(* CODESYS project SingleElevator.project

Project tree, tasks and I/O mapping:
  Device : CODESYS Control Win V3, 3S - Smart Software Solutions GmbH, version 3.5.16.20
    application Application
      libraries: Standard, * (System)
      task MainTask (cyclic, interval t#20ms, priority 1) calls Simulation, GAinstances, PLC_PRG
      task VISU_TASK (cyclic, interval 100 ms, priority 31) calls VisuElems.Visu_Prg
      global variables GVL
      visualisation Visualization
      program Simulation [ST]
      program GAinstances [FBD]
      program PLC_PRG [SFC]: Closing_active, Closing_exit, CloseDoors2_exit, CloseDoors_active, CloseDoors_exit, FirstFloor_active, FirstFloor_exit, OpenDoors_active, OpenDoors_exit, CloseDoors2_active, Destination_active, Destination_exit, OpenDoors2_active, OpenDoors2_exit, WaitForCalls_active, PreCalls_active, MidCalls_active, MidCalls_entry, WaitForCalls_exit, PreCalls_entry, Dummy4_exit, LEDActive_active, LEDnotActive_active, GetCalls_active, FirstFloor_entry, Destination_entry
      GA/
        function block Doors_GA [SFC]: Init_active, Ready_active, Busy_active
        function block Motoring_GA [SFC]: Init_active, Ready_active, Busy_active, StartMotor_active, HighSpeed_active, StartGoDown_active, StartGoDown_exit, GroundFloor_active, GroundFloor_exit, LowSpeed_active, LowSpeed_exit, CountingDecks_active, Working_active, Extremes_active, Extremes_exit, Extremes_entry, StartMotor_exit
  text list GlobalTextList
*)

// Device/Application/GVL
{attribute 'qualified_only'}
VAR_GLOBAL
	ManageDoors: Doors_GA;
	Motoring : Motoring_GA;
	
(* Elevator managing variables*)
	Open: BOOL;				(* Sensor: the door is fully open*)
	Closed: BOOL;			(* Sensor: the door is fully closed*)
	LimitDown: BOOL;		(* Sensor: lower limit sensor, if TRUE the lift has reached the lower limit*)
	LimitUp: BOOL;			(* Sensor: upper limit sensor, if TRUE the lift has reached the upper limit*)
	DeckSensor: BOOL;		(* Sensor: if TRUE the cab is in proximity of a deck*)
	RampSensor: BOOL;		(* Sensor: if TRUE the cab is in proximity of a ramp*)
	Presence :BOOL; 		(* Sensor: if TRUE something blocks the door photocell*)
	Emergency: BOOL;		(* Input: if TRUE the emergency button has been pressed*)

	Closing: BOOL;			(* Actuator: if TRUE the door starts closing*)
	Opening: BOOL;			(* Actuator: the door starts opening*)
	Motor_on: BOOL;			(* Actuator: if TRUE the lift pulley motor start moving*)
	Up: BOOL;				(* Actuator parameter: if TRUE the lift moves upward, downward otherwise*)
	Vel: BOOL;				(* Actuator parameter: motor speed, if TRUE high speed, low speed otherwise*)


	Current: INT;  			(* Visualization: variable used to storage the current deck*)
    Destination: INT;		(* Visualization: variable used to storage the the destination deck*)
	EmergencyVis: BOOL; 	(* Visualization: if TRUE the emergency light is turned on*)

	InitialDeck: INT := 1;	(* Only for simulation: variable used to define the initial deck*)
	InitCycle: BOOL := FALSE;(* Only for simulation: used to execute the instruction at the first cycle*)
	Height: INT;			(* Only for simulation: elevator height*)
	DeckRest: INT;        	(* Only for simulation: division rest for generating deck sensor*)
	Memory: INT;
	RampRest: INT;			(* Only for simulation: division rest for generating the ramp position*)
	MemoryR: INT;
	Door: INT;				(* Only for simulation: to visualize the closing of the door*)
	Displacement: INT;		(* Only for simulation: lift displacement, dependent on the motor speed*)

 (*Inputs: internal panel variables*)
	PG: BOOL;
	P1: BOOL;
	P2: BOOL;
	P3: BOOL;
	P4: BOOL;
	P5: BOOL;
	P6: BOOL;
	P7: BOOL;

(*Visualization: internal panel variables used to turn on the LED*)
	PGVis: BOOL;
	P1Vis: BOOL;
	P2Vis: BOOL;
	P3Vis: BOOL;
	P4Vis: BOOL;
	P5Vis: BOOL;
	P6Vis: BOOL;
	P7Vis: BOOL;

(*Inputs: external panel variables*)
	UpDeckG: BOOL;
	UpDeck1: BOOL;
	UpDeck2: BOOL;
	UpDeck3: BOOL;
	UpDeck4: BOOL;
	UpDeck5: BOOL;
	UpDeck6: BOOL;
	DownDeck7: BOOL;
	DownDeck6: BOOL;
	DownDeck5: BOOL;
	DownDeck4: BOOL;
	DownDeck3: BOOL;
	DownDeck2: BOOL;
	DownDeck1: BOOL;

(*Visualization: external panel variables used to turn on the LED*)
	UpDeckGVis: BOOL;
	UpDeck1Vis: BOOL;
	UpDeck2Vis: BOOL;
	UpDeck3Vis: BOOL;
	UpDeck4Vis: BOOL;
	UpDeck5Vis: BOOL;
	UpDeck6Vis: BOOL;
	DownDeck7Vis: BOOL;
	DownDeck6Vis: BOOL;
	DownDeck5Vis: BOOL;
	DownDeck4Vis: BOOL;
	DownDeck3Vis: BOOL;
	DownDeck2Vis: BOOL;
	DownDeck1Vis: BOOL;

(*Only for simulation: variables used to simulate the fault on deck sensor*)
	SensorG: BOOL;				(* if TRUE the magnetic information for deck G is lost and the deck sensor cannot become TRUE*)
	Sensor1: BOOL;				(* if TRUE the magnetic information for deck 1 is lost and the deck sensor cannot become TRUE*)
	Sensor2: BOOL;
	Sensor3: BOOL;
	Sensor4: BOOL;
	Sensor5: BOOL;
	Sensor6: BOOL;
	Sensor7: BOOL;
	FaultSensorAlarm: BOOL; 	(* Visulaization: if TRUE alerts the user of a deck sensor fault*)

(*Only for simulation: variables used to simulate the fault on ramp sensor*)
	RampGUp: BOOL;
	Ramp1Down: BOOL;
	Ramp1Up:BOOL;
	Ramp2Down: BOOL;
	Ramp2Up:BOOL;
	Ramp3Down: BOOL;
	Ramp3Up:BOOL;
	Ramp4Down: BOOL;
	Ramp4Up:BOOL;
	Ramp5Down: BOOL;
	Ramp5Up:BOOL;
	Ramp6Down: BOOL;
	Ramp6Up:BOOL;
	Ramp7Down: BOOL;
	FaultRampAlarm: BOOL; 		(* Visulaization: if TRUE alerts the user of a ramp sensor fault*)
	SensorGOK: BOOL;
	Sensor1OK: BOOL;
	Sensor2OK: BOOL;
	Sensor6OK: BOOL;
	Sensor3OK: BOOL;
	Sensor4OK: BOOL;
	Sensor5OK: BOOL;
	Sensor7OK: BOOL;
	RampGUpOK: BOOL;
	Ramp1DownOK: BOOL;
	Ramp1UpOK: BOOL;
	Ramp2DownOK: BOOL;
	Ramp2UpOK: BOOL;
	Ramp3DownOK: BOOL;
	Ramp3UpOK: BOOL;
	Ramp4DownOK: BOOL;
	Ramp4UpOK: BOOL;
	Ramp5DownOK: BOOL;
	Ramp5UpOK: BOOL;
	Ramp6DownOK: BOOL;
	Ramp6UpOK: BOOL;
	Ramp7DownOK: BOOL;
	Ramp7UpOK: BOOL;
END_VAR

// Device/Application/Simulation
PROGRAM Simulation
VAR
END_VAR

(* Initial position of the cab inside the hoistway. It is executed only at the first cycle.  *)
IF NOT GVL.InitCycle THEN
			GVL.InitCycle := TRUE ;
			GVL.Height := 20 * GVL.InitialDeck;
		    GVL.Door := 0;
			GVL.Current := GVL.Height / 20;
END_IF;

(* Elevator management, these instructions are executed each cycle time*)

(* Elevator door control. *)
IF GVL.Closing THEN
	GVL.Door := GVL.Door + 1;		(*Closing door management*)
	GVL.Open := FALSE;
END_IF

IF GVL.Door >= 60 THEN						(* Closed door limit*)
	GVL.Closed := TRUE;
END_IF

IF GVL.Opening THEN
	GVL.Door := GVL.Door - 1; 	(* Opening door management*)
	GVL.Closed := FALSE;
END_IF

IF GVL.Door <= 0 THEN							(* Open door limit*)
	GVL.Open := TRUE;
END_IF


(* Maximum and minimum management in the door simulation*)
IF GVL.Door < 0 THEN
	 GVL.Door := 0;
END_IF

IF GVL.Door > 60 THEN
	GVL.Door := 60;
END_IF


(* Control of the cab position inside the hostway. *)
(* Displacement definition for graphic visualization*)
IF GVL.Vel THEN 
	GVL.Displacement := 2;
ELSE 
	GVL.Displacement := 1;
END_IF


(* Height modification relying on direction and speed*)
IF GVL.Motor_on AND GVL.Up THEN
	GVL.Height := GVL.Height + GVL.Displacement;
	GVL.LimitDown := FALSE;
END_IF

IF GVL.Motor_on AND NOT GVL.Up THEN
	GVL.Height := GVL.Height - GVL.Displacement;
	GVL.LimitUp := FALSE;
END_IF


(* Limits for visualization*)
IF GVL.Height < -20 THEN
	GVL.Height := -20;
END_IF

IF GVL.Height > 160 THEN
	GVL.Height := 160;
END_IF

(* Limit sensors management*)
IF GVL.Height <= -10 THEN
	GVL.LimitDown := TRUE;
END_IF

IF GVL.Height >= 150 THEN
	 GVL.LimitUp := TRUE;
END_IF


(*-------------------------------------------------------------------*)
(*  Fault Management (Deck and Ramp Sensors)   *)
(*-------------------------------------------------------------------*)
(* Deck Sensor*)
(* Range of value where the deck sensor is active*)
IF ((GVL.Height >= -1) AND (GVL.Height <= 1)) THEN
	GVL.SensorGOK := TRUE;
ELSE  
	GVL.SensorGOK := FALSE;
END_IF

IF ((GVL.Height >= 20-1) AND (GVL.Height <= 20+1)) THEN
	GVL.Sensor1OK := TRUE;
ELSE  
	GVL.Sensor1OK := FALSE;
END_IF

IF ((GVL.Height >= 40-1) AND (GVL.Height <= 40+1)) THEN
	GVL.Sensor2OK := TRUE;
ELSE  
	GVL.Sensor2OK := FALSE;
END_IF

IF ((GVL.Height >= 60-1) AND (GVL.Height <= 60+1)) THEN
	GVL.Sensor3OK := TRUE;
ELSE  
	GVL.Sensor3OK := FALSE;
END_IF

IF ((GVL.Height >= 80-1) AND (GVL.Height <= 80+1)) THEN
	GVL.Sensor4OK := TRUE;
ELSE  
	GVL.Sensor4OK := FALSE;
END_IF

IF ((GVL.Height >= 100-1) AND (GVL.Height <= 100+1)) THEN
	GVL.Sensor5OK := TRUE;
ELSE   
	GVL.Sensor5OK := FALSE;
END_IF

IF ((GVL.Height >= 120-1) AND (GVL.Height <= 120+1)) THEN
	GVL.Sensor6OK := TRUE;
ELSE  
	GVL.Sensor6OK := FALSE;
END_IF

IF ((GVL.Height >= 140-1) AND (GVL.Height <= 140+1)) THEN
	GVL.Sensor7OK := TRUE;
ELSE  
	GVL.Sensor7OK := FALSE;
END_IF

GVL.DeckSensor := (GVL.SensorGOK AND NOT GVL.SensorG) OR
				    (GVL.Sensor1OK AND NOT GVL.Sensor1) OR
				    (GVL.Sensor2OK AND NOT GVL.Sensor2) OR
				    (GVL.Sensor3OK AND NOT GVL.Sensor3) OR
				    (GVL.Sensor4OK AND NOT GVL.Sensor4) OR
				    (GVL.Sensor5OK AND NOT GVL.Sensor5) OR
				    (GVL.Sensor6OK AND NOT GVL.Sensor6) OR
				    (GVL.Sensor7OK AND NOT GVL.Sensor7);

(* Ramp Sensor*)
(* Range of value where the ramp sensor is active*)
IF ((GVL.Height >= 5-1) AND (GVL.Height <= 5+1)) THEN
	GVL.RampGUpOK := TRUE;
ELSE 
	GVL.RampGUpOK := FALSE;
END_IF

(* Ramp close to deck 1*)
IF ((GVL.Height >= 15-1) AND (GVL.Height <= 15+1)) THEN
	GVL.Ramp1DownOK := TRUE;
ELSE 
	GVL.Ramp1DownOK := FALSE;
END_IF

IF ((GVL.Height >= 25-1) AND (GVL.Height <= 25+1)) THEN
	GVL.Ramp1UpOK := TRUE;
ELSE 
	GVL.Ramp1UpOK := FALSE;
END_IF

(* Ramp close to deck 2*)
IF ((GVL.Height >= 35-1) AND (GVL.Height <= 35+1)) THEN
	GVL.Ramp2DownOK := TRUE;
ELSE 
	GVL.Ramp2DownOK := FALSE;
END_IF

IF ((GVL.Height >= 45-1) AND (GVL.Height <= 45+1)) THEN
	GVL.Ramp2UpOK := TRUE;
ELSE 
	GVL.Ramp2UpOK := FALSE;
END_IF

(*Ramp close to deck  3*)
IF ((GVL.Height >= 55-1) AND (GVL.Height <= 55+1)) THEN
	GVL.Ramp3DownOK := TRUE;
ELSE 
	GVL.Ramp3DownOK := FALSE;
END_IF

IF ((GVL.Height >= 65-1) AND (GVL.Height <= 65+1)) THEN
	GVL.Ramp3UpOK := TRUE;
ELSE 
	GVL.Ramp3UpOK := FALSE;
END_IF

(* Ramp close to deck  4*)
IF ((GVL.Height >= 75-1) AND (GVL.Height <= 75+1)) THEN
	GVL.Ramp4DownOK := TRUE;
ELSE 
	GVL.Ramp4DownOK := FALSE;
END_IF

IF ((GVL.Height >= 85-1) AND (GVL.Height <= 85+1)) THEN
	GVL.Ramp4UpOK := TRUE;
ELSE 
	GVL.Ramp4UpOK:=FALSE;
END_IF

(* Ramp close to deck  5*)
IF ((GVL.Height >= 95-1) AND (GVL.Height <= 95+1)) THEN
	GVL.Ramp5DownOK := TRUE;
ELSE 
	GVL.Ramp5DownOK := FALSE;
END_IF

IF ((GVL.Height >= 105-1) AND (GVL.Height <= 105+1)) THEN
	GVL.Ramp5UpOK := TRUE;
ELSE
	GVL.Ramp5UpOK := FALSE;
END_IF

(* Ramp close to deck  6*)
IF ((GVL.Height >= 115-1) AND (GVL.Height <= 115+1)) THEN
	GVL.Ramp6DownOK := TRUE;
ELSE 
	GVL.Ramp6DownOK := FALSE;
END_IF

IF ((GVL.Height >= 125-1) AND (GVL.Height <= 125+1)) THEN
	GVL.Ramp6UpOK := TRUE;
ELSE 
	GVL.Ramp6UpOK := FALSE;
END_IF

(* Ramp close to deck  7*)
IF ((GVL.Height >= 135-1) AND (GVL.Height <= 135+1)) THEN
	GVL.Ramp7DownOK := TRUE;
ELSE 
	GVL.Ramp7DownOK := FALSE;
END_IF

GVL.RampSensor:=(GVL.RampGUpOK AND NOT GVL.RampGUp) OR 
								(GVL.Ramp1DownOK AND NOT GVL.Ramp1Down ) OR 
								(GVL.Ramp1UpOK AND NOT GVL.Ramp1Up ) OR
								(GVL.Ramp2DownOK AND NOT GVL.Ramp2Down ) OR 
								(GVL.Ramp2UpOK AND NOT GVL.Ramp2Up ) OR
								(GVL.Ramp3DownOK AND NOT GVL.Ramp3Down ) OR
 								(GVL.Ramp3UpOK AND NOT GVL.Ramp3Up ) OR
								(GVL.Ramp4DownOK AND NOT GVL.Ramp4Down ) OR
 								(GVL.Ramp4UpOK AND NOT GVL.Ramp4Up ) OR
								(GVL.Ramp5DownOK AND NOT GVL.Ramp5Down ) OR
 								(GVL.Ramp5UpOK AND NOT GVL.Ramp5Up ) OR
								(GVL.Ramp6DownOK AND NOT GVL.Ramp6Down ) OR
								(GVL.Ramp6UpOK AND NOT GVL.Ramp6Up ) OR
								(GVL.Ramp7DownOK AND NOT GVL.Ramp7Down );

END_PROGRAM

// Device/Application/GAinstances
PROGRAM GAinstances
VAR
END_VAR

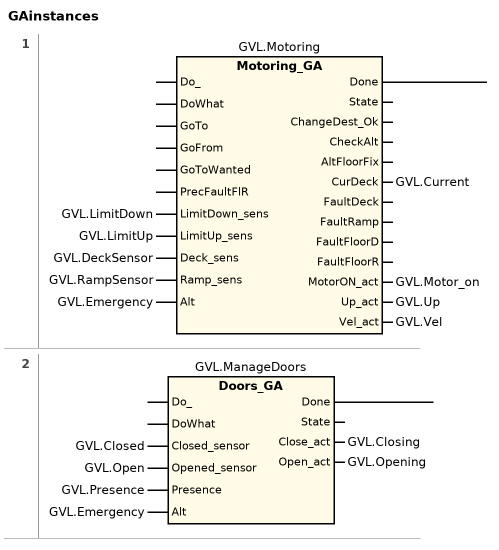
// NETWORK 1
GVL.Motoring(
    LimitDown_sens := GVL.LimitDown,
    LimitUp_sens := GVL.LimitUp,
    Deck_sens := GVL.DeckSensor,
    Ramp_sens := GVL.RampSensor,
    Alt := GVL.Emergency,
    CurDeck => GVL.Current,
    MotorON_act => GVL.Motor_on,
    Up_act => GVL.Up,
    Vel_act => GVL.Vel); // Motoring_GA

// NETWORK 2
GVL.ManageDoors(
    Closed_sensor := GVL.Closed,
    Opened_sensor := GVL.Open,
    Presence := GVL.Presence,
    Alt := GVL.Emergency,
    Close_act => GVL.Closing,
    Open_act => GVL.Opening); // Doors_GA

END_PROGRAM

// Device/Application/GA/Motoring_GA
FUNCTION_BLOCK Motoring_GA
VAR_INPUT
	Do_: BOOL;
	DoWhat: STRING;
	GoTo: INT;
	GoFrom: INT;
	GoToWanted: INT;
	PrecFaultFlR: ARRAY[0..7] OF INT;
	
	//SENSORS
	LimitDown_sens: BOOL;
	LimitUp_sens: BOOL;
	Deck_sens: BOOL;
	Ramp_sens: BOOL;
	
	Alt: BOOL;
END_VAR

VAR_OUTPUT
	Done: BOOL;
	State: STRING;
	ChangeDest_Ok: BOOL;
	CheckAlt: BOOL;
	AltFloorFix: INT;
	CurDeck: INT;
	
	//FAULTS
	FaultDeck: BOOL;
	FaultRamp: BOOL;
	FaultFloorD: ARRAY[0..7] OF INT;
	FaultFloorR: ARRAY[0..7] OF INT;
	
	//ACTUATORS
	MotorON_act: BOOL;
	Up_act: BOOL;
	Vel_act: BOOL;
END_VAR
VAR
	i: INT;
	Cont: INT;
	CheckRamps: BOOL;
	Initial: BOOL;
	
	AltFloor: INT;
	Fault: BOOL;
	Faults: ARRAY[0..21] OF BOOL;
	DeckPrec: INT;
	RampPrec: INT;
	FirstTime: BOOL;
	TrueFault: INT;
	NoProbFault: BOOL;
	FaultSameD: BOOL;
	SecondRamp: BOOL;
	Down_sens: BOOL;
	Up_sens: BOOL;
	CorrDone: BOOL;
	Sens: BOOL;
END_VAR

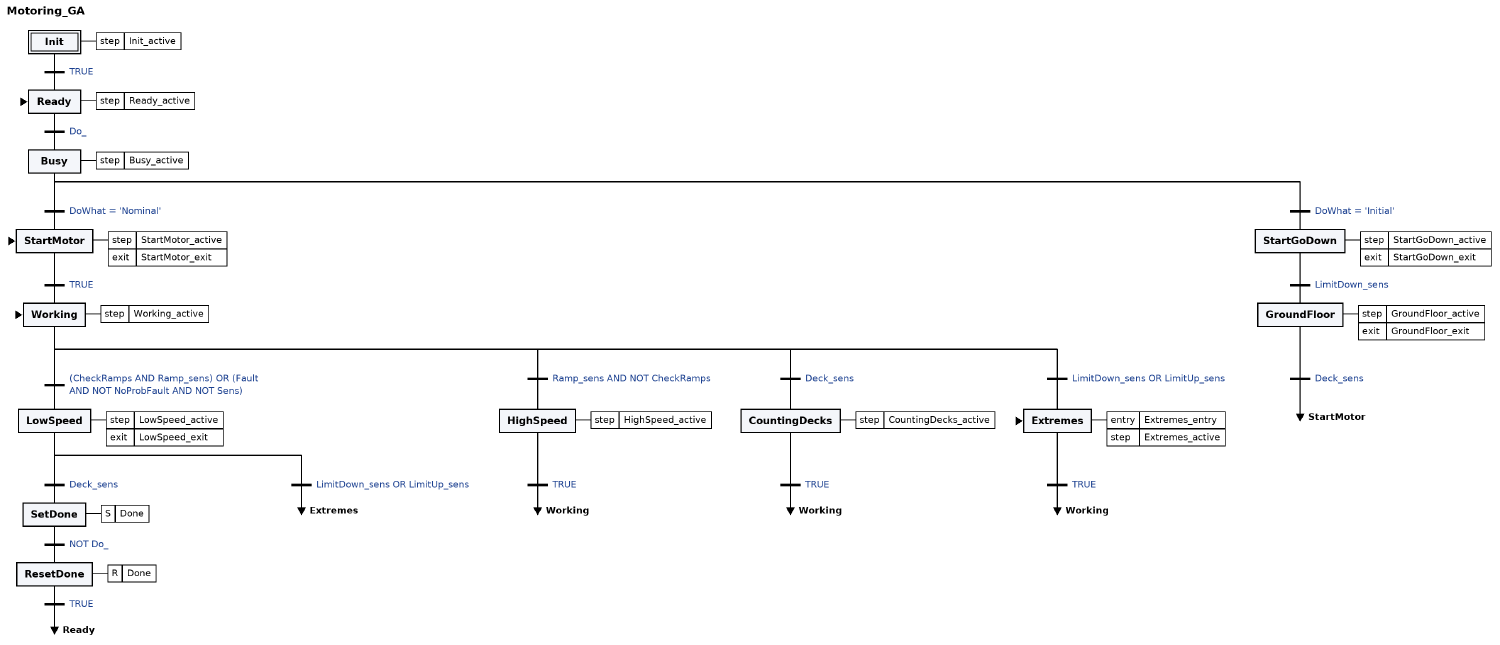
INITIAL_STEP Init:
    Init_active(N);  // step action
END_STEP
TRANSITION FROM Init TO Ready
    := TRUE;
END_TRANSITION
STEP Ready:
    Ready_active(N);  // step action
END_STEP
TRANSITION FROM Ready TO Busy
    := Do_;
END_TRANSITION
STEP Busy:
    Busy_active(N);  // step action
END_STEP
TRANSITION FROM Busy TO StartMotor
    := DoWhat = 'Nominal';
END_TRANSITION
STEP StartMotor:
    StartMotor_active(N);  // step action
    StartMotor_exit(P0);  // exit action
END_STEP
TRANSITION FROM StartMotor TO Working
    := TRUE;
END_TRANSITION
STEP Working:
    Working_active(N);  // step action
END_STEP
TRANSITION FROM Working TO LowSpeed
    := (CheckRamps AND Ramp_sens) OR (Fault AND NOT NoProbFault AND NOT Sens);
END_TRANSITION
STEP LowSpeed:
    LowSpeed_active(N);  // step action
    LowSpeed_exit(P0);  // exit action
END_STEP
TRANSITION FROM Working TO HighSpeed
    := Ramp_sens AND NOT CheckRamps;
END_TRANSITION
STEP HighSpeed:
    HighSpeed_active(N);  // step action
END_STEP
TRANSITION FROM HighSpeed TO Working
    := TRUE;
END_TRANSITION
TRANSITION FROM Working TO CountingDecks
    := Deck_sens;
END_TRANSITION
STEP CountingDecks:
    CountingDecks_active(N);  // step action
END_STEP
TRANSITION FROM CountingDecks TO Working
    := TRUE;
END_TRANSITION
TRANSITION FROM Working TO Extremes
    := LimitDown_sens OR LimitUp_sens;
END_TRANSITION
STEP Extremes:
    Extremes_entry(P1);  // entry action
    Extremes_active(N);  // step action
END_STEP
TRANSITION FROM Extremes TO Working
    := TRUE;
END_TRANSITION
TRANSITION FROM LowSpeed TO SetDone
    := Deck_sens;
END_TRANSITION
TRANSITION FROM LowSpeed TO Extremes
    := LimitDown_sens OR LimitUp_sens;
END_TRANSITION
TRANSITION FROM Busy TO StartGoDown
    := DoWhat = 'Initial';
END_TRANSITION
STEP StartGoDown:
    StartGoDown_active(N);  // step action
    StartGoDown_exit(P0);  // exit action
END_STEP
TRANSITION FROM StartGoDown TO GroundFloor
    := LimitDown_sens;
END_TRANSITION
STEP GroundFloor:
    GroundFloor_active(N);  // step action
    GroundFloor_exit(P0);  // exit action
END_STEP
TRANSITION FROM GroundFloor TO StartMotor
    := Deck_sens;
END_TRANSITION
STEP SetDone:
    Done(S);
END_STEP
TRANSITION FROM SetDone TO ResetDone
    := NOT Do_;
END_TRANSITION
STEP ResetDone:
    Done(R);
END_STEP
TRANSITION FROM ResetDone TO Ready
    := TRUE;
END_TRANSITION

ACTION Init_active:
State:='Init';
END_ACTION

ACTION Ready_active:
State:='Ready';
END_ACTION

ACTION Busy_active:
State:='Busy';
END_ACTION

ACTION StartMotor_active:
//Set correct motion direction
IF (GoTo - GoFrom) > 0 THEN
	Up_act := TRUE;
ELSE
	Up_act := FALSE;
END_IF

//The motors starts moving at LOW speed
Vel_act := FALSE;
MotorON_act := TRUE;
END_ACTION

ACTION HighSpeed_active:
//Ramp counter
Cont := Cont + 1;

//Checking the path that require HIGH Speed
IF Cont = ABS(GoTo - GoFrom)*2 -1 THEN
	CheckRamps := TRUE;
END_IF

//If Initializing, Speed is always set to LOW
IF NOT Initial THEN
	Vel_act := TRUE;
END_IF

//Checking if it is possible to change destination mid-functioning 
//It is checked if New Destination is reachable at LOW Speed
IF (Up_act AND (GotoWanted <> -1) AND
	(GoToWanted > CurDeck + (Cont MOD 2) - 1) AND
	Cont < ABS(GoToWanted - GoFrom)*2 - 1) THEN 
	
	ChangeDest_Ok := TRUE;
	
ELSIF (NOT Up_act AND (GotoWanted <> -1) AND
	(GoToWanted < CurDeck - (Cont MOD 2) + 1) AND
	Cont < ABS(GoToWanted - GoFrom)*2 - 1) THEN
	
	ChangeDest_Ok := TRUE;
	
END_IF

//EMERGENCY HANDLING
//In case of Emergency, the elevator finds the nearest 'safe' floor to stop at
IF Alt THEN
	//Here the 'safe' floor is found
	FOR i := 0 TO 7 BY 1 DO
		IF Up_act AND ((7-i) > CurDeck + (Cont MOD 2) - 1) AND
			Cont < ABS((7-i) - GoFrom)*2 - 1 THEN
			AltFloor := 7 - i;
		ELSIF NOT Up_act AND (i < CurDeck - (Cont MOD 2) + 1) AND
			Cont < ABS(i - GoFrom)*2 - 1 THEN
			AltFloor := i;
		END_IF
	END_FOR
	//The floor is saved and sent as output to the Policy
	IF AltFloor <> -1 AND NOT CheckAlt THEN
		AltFloorFix := AltFloor;  
		CheckAlt := TRUE;
	END_IF
END_IF
END_ACTION

ACTION StartGoDown_active:
//Setting LOW speed motion DOWNWARDS for Initialization
Initial := TRUE;
Up_act := FALSE;
Vel_act := FALSE;
MotorON_act := TRUE;
END_ACTION

ACTION StartGoDown_exit:
MotorON_act := FALSE;
END_ACTION

ACTION GroundFloor_active:
//Once reached the Down Limit, the elevator reaches Ground floor
Up_act := TRUE;
MotorON_act := TRUE;
END_ACTION

ACTION GroundFloor_exit:
MotorON_act := FALSE;
END_ACTION

ACTION LowSpeed_active:
//Speed from now on is set to LOW
Vel_act := FALSE;

//Detection of a problematic Deck Fault and its associated Fault Floor
//A correction is made to the direction if extremes are detected
IF Ramp_sens AND NOT NoProbFault AND SecondRamp AND NOT Initial THEN
	IF ((Up_act AND NOT Down_sens) OR Up_sens) AND PrecFaultFlR[0] <> GoTo THEN
		FaultDeck := TRUE;
		FaultFloorD[0] := (i+1)/3;
	END_IF
	IF((NOT Up_act AND NOT Up_sens) OR Down_sens) AND PrecFaultFlR[1] <> GoTo THEN
		FaultDeck := TRUE;
		FaultFloorD[0] := (CurDeck-Cont+GoFrom*2)/3;
	END_IF
END_IF

//Two Ramps are needed to make the code above work
IF Ramp_sens THEN
	SecondRamp := TRUE;
END_IF
END_ACTION

ACTION LowSpeed_exit:
//Current Deck Correction - Always performed
IF Up_act THEN
	CurDeck := CurDeck + 1;
ELSE
	CurDeck := CurDeck - 1;
END_IF

//Current Deck Correction - Extremes detected
IF Down_sens THEN
	CurDeck := CurDeck - 1;
END_IF
IF Up_sens THEN
	CurDeck := CurDeck + 1;
END_IF

//Fault Floor Correction (1) - Starting Floor Deck Fault
IF FaultSameD AND FaultFloorD[0] <> -1 THEN
	IF Up_act THEN
		FaultFloorD[0] := FaultFloorD[0] - 1;
	ELSE
		FaultFloorD[0] := FaultFloorD[0] + 1;
	END_IF
END_IF

//Current Deck Correction - Generic Deck Fault
IF FaultDeck THEN
	IF Up_act THEN
		CurDeck := CurDeck + 1;
	ELSE
		CurDeck := CurDeck - 1;
	END_IF
END_IF

//Fault Floor Correction (2) - Starting Floor Deck Fault
IF FaultSameD AND FaultFloorD[0] = -1 THEN
	FaultDeck := TRUE;
	FaultFloorD[0] := GoFrom;
END_IF

Fault := FaultDeck OR FaultRamp; //Fault is a generic Fault
ChangeDest_OK := FALSE; //Reset possible destination change
Initial := FALSE; //Reset initialization variable
MotorON_act := FALSE; //Motor is turned OFF once the last Deck is detected
END_ACTION

ACTION CountingDecks_active:
//Here the Deck counter is implemented
IF Up_act AND FirstTime THEN
	CurDeck := CurDeck + 1;
ELSIF NOT Up_act AND FirstTime THEN
	CurDeck := CurDeck - 1;
END_IF
//The first Deck does not have to be counted
FirstTime := TRUE;
END_ACTION

ACTION Working_active:
//In this block, Ramp_sens and Deck_sens states are stored and analysed

//Filling a Boolean Array with Ramp and Deck sequence
//Ramp Sensor -> FALSE
//Deck Sensor -> TRUE

IF Up_act AND NOT (Down_sens OR Up_sens) THEN
	IF DeckPrec <> CurDeck THEN 
		DeckPrec := CurDeck;
		Faults[CurDeck+Cont+GoFrom*2] := TRUE;
	END_IF
	IF RampPrec <> Cont THEN
		RampPrec := Cont;
		Faults[CurDeck+Cont+GoFrom*2] := FALSE;
	END_IF
ELSIF NOT Up_act AND NOT (Down_sens OR Up_sens) THEN
	IF DeckPrec <> CurDeck THEN 
		DeckPrec := CurDeck;
		Faults[CurDeck-Cont+GoFrom*2] := TRUE;
	END_IF
	IF RampPrec <> Cont THEN
		RampPrec := Cont;
		Faults[CurDeck-Cont+GoFrom*2] := FALSE;
	END_IF
END_IF

//Detection of a Fault Deck at the starting Floor
IF NOT FirstTime AND Cont = 1 THEN
	FaultSameD := TRUE;
END_IF

//Management of an already detected Ramp Fault
IF Up_act AND PrecFaultFlR[1] >= GoFrom AND PrecFaultFlR[0] <= GoTo AND CurDeck = PrecFaultFlR[1] AND NOT CorrDone THEN
	IF PrecFaultFlR[0] = GoTo THEN
		Checkramps := TRUE;
	ELSE
		Cont := Cont + 1; //Adding the 'missing' Ramp
	END_IF
	CorrDone := TRUE;
ELSIF NOT Up_act AND PrecFaultFlR[0] <= GoFrom AND PrecFaultFlR[1] >= GoTo AND CurDeck = PrecFaultFlR[0] AND NOT CorrDone THEN
	IF PrecFaultFlR[1] = GoTo THEN
		Checkramps := TRUE;
	ELSE
		Cont := Cont + 1; //Adding the 'missing' Ramp
	END_IF
	CorrDone := TRUE;
END_IF

//Looking for Faults in the Ramp/Deck sequence Array
//Subdividing them in two groups: FaultDeck and FaultRamp
IF Up_act AND NOT (Down_sens OR Up_sens) THEN
	FOR i := GoFrom*3+1 TO CurDeck+Cont+GoFrom*2 BY 1 DO
		IF (i MOD 3) = 0 AND Faults[i] <> TRUE AND (NOT FaultDeck AND NOT FaultRamp) THEN
			FaultDeck := TRUE;
			FaultFloorD[0] := i/3;
		END_IF
		IF (i MOD 3) <> 0 AND Faults[i] <> FALSE AND (NOT FaultDeck AND NOT FaultRamp) THEN
			FaultRamp := TRUE;
			FaultFloorR[0] := (i+1)/3;
			FaultFloorR[1] := (i-2)/3;
		END_IF
	END_FOR
ELSIF NOT Up_act AND NOT (Down_sens OR Up_sens) THEN
	FOR i := CurDeck-Cont+GoFrom*2 TO GoFrom*3-1 BY 1 DO
		IF (i MOD 3) = 0 AND Faults[i] <> TRUE AND (NOT FaultDeck AND NOT FaultRamp) THEN
			FaultDeck := TRUE;
			FaultFloorD[0] := i/3;
		END_IF
		IF (i MOD 3) <> 0 AND Faults[i] <> FALSE AND (NOT FaultDeck AND NOT FaultRamp) THEN
			FaultRamp := TRUE;
			FaultFloorR[0] := (i+2)/3;
			FaultFloorR[1] := (i-1)/3;
		END_IF
	END_FOR
END_IF

Fault := FaultDeck OR FaultRamp; //Fault is a generic Fault

//Checking if a Fault is not 'problematic'
//A problematic Fault is a Fault that doesn't allow to stop at the desired destination
//If the Fault is problematic the speed is set to LOW
IF Up_act AND (FaultFloorD[0] <> GoTo AND FaultFloorD[0] <> -1) OR (FaultFloorR[0] <> GoTo AND FaultFloorR[0] <> -1) AND NOT NoProbFault THEN
	NoProbFault := TRUE;
	IF FaultRamp AND PrecFaultFlR[1] = -1 THEN
		Cont := Cont + 1;
	END_IF
ELSIF NOT Up_act AND (FaultFloorD[0] <> GoTo AND FaultFloorD[0] <> -1) OR (FaultFloorR[1] <> GoTo AND FaultFloorR[1] <> -1) AND NOT NoProbFault THEN
	NoProbFault := TRUE;
	IF FaultRamp AND PrecFaultFlR[1] = -1 THEN
		Cont := Cont + 1;
	END_IF
END_IF

Sens := Ramp_sens OR Deck_sens OR LimitDown_sens OR LimitUp_sens; //For mutual exclusion purposes
END_ACTION

ACTION Extremes_active:
//Stop motor
MotorON_act := FALSE;

//Reverse direction
IF Down_sens THEN
	Up_act := TRUE;
ELSIF Up_sens THEN
	Up_act := FALSE;
END_IF

//Start motor again
MotorON_act := TRUE;
END_ACTION

ACTION Extremes_exit:

END_ACTION

ACTION Extremes_entry:
//Storing if Extremes are reached
IF NOT Down_sens THEN
	Down_sens := LimitDown_sens;
END_IF
IF NOT Up_sens THEN
	Up_sens := LimitUp_sens;
END_IF
END_ACTION

ACTION StartMotor_exit:
//Variables Initialization

CurDeck := GoFrom; //Current Deck
Cont := 0; //Ramp counter
CheckRamps := FALSE; //If TRUE we have to set LOW speed at next Ramp
FirstTime := FALSE; //Ensure that Deck corrections are done once

GoToWanted := -1; //Alternative desired destination 
ChangeDest_Ok := FALSE; //If TRUE we can change destination mid-functioning

AltFloor:= -1; //Nearest Floor destination when Emergency is ON
CheckAlt:= FALSE; //To fix AltFloor value

DeckPrec := CurDeck; //Contains the previous Deck value
RampPrec := Cont; //Contains the previous Ramp value

FaultDeck := FALSE; //Detects if a Deck Fault is present
FaultRamp := FALSE; //Detects if a Ramp Fault is present
Fault := FALSE; //Detects if any kind of Fault is present
NoProbFault := FALSE; //Detects if a Fault is 'problematic'
FaultSameD := FALSE; //Detects if a Deck Fault happens at the starting Floor 
SecondRamp := FALSE; //Verifies if there is a 'problematic' Deck Fault
Down_sens := FALSE; //Keeps the TRUE value of LimitDown_sens
Up_sens := FALSE; //Keeps the TRUE value of LimitUp_sens
Sens := FALSE; //Detects if any sensor is true
CorrDone := FALSE; //Ensure the correction when there is a Ramp Fault

FOR i := 0 TO 21 BY 1 DO
	Faults[i] := FALSE; //Array that stores Ramp/Deck sequence
END_FOR

FOR i := 0 TO 7 BY 1 DO
	FaultFloorD[i] := -1; //Array that stores Deck Faults
	FaultFloorR[i] := -1; //Array that stores Ramp Faults
END_FOR
END_ACTION

END_FUNCTION_BLOCK

// Device/Application/GA/Doors_GA
FUNCTION_BLOCK Doors_GA
VAR_INPUT
	Do_: BOOL;
	DoWhat: STRING;
	
	//SENSORS
	Closed_sensor: BOOL;
	Opened_sensor: BOOL;
	Presence : BOOL;
	
	Alt: BOOL;
END_VAR
VAR_OUTPUT
	Done: BOOL;
	State: STRING;
	
	//ACTUATORS
	Close_act: BOOL;
	Open_act: BOOL;
END_VAR
VAR
END_VAR

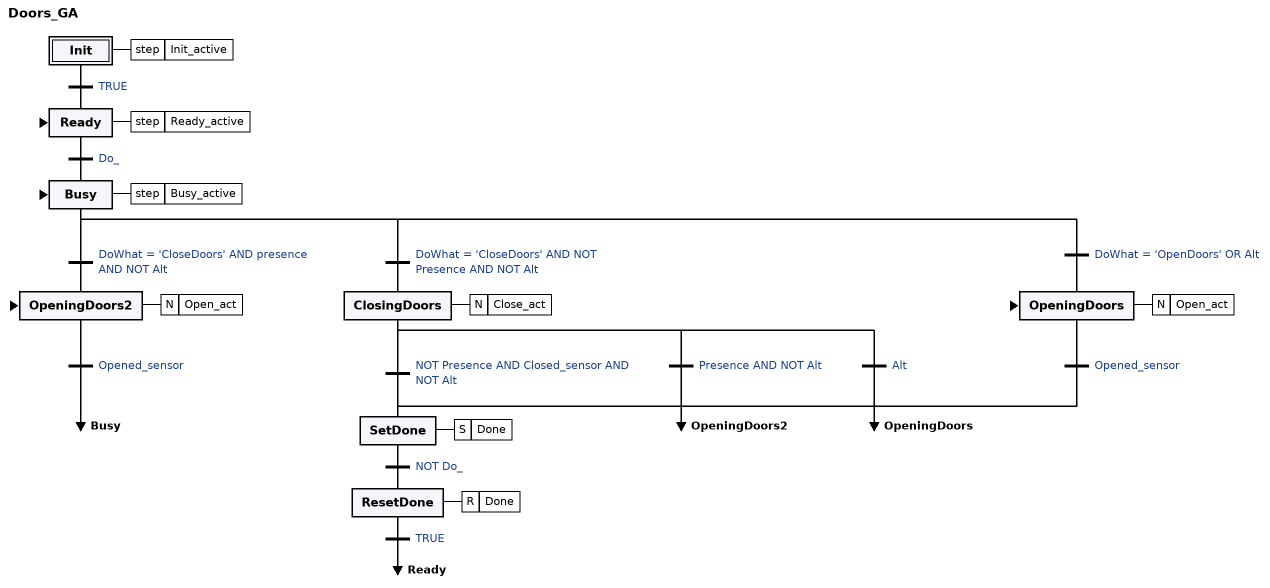
INITIAL_STEP Init:
    Init_active(N);  // step action
END_STEP
TRANSITION FROM Init TO Ready
    := TRUE;
END_TRANSITION
STEP Ready:
    Ready_active(N);  // step action
END_STEP
TRANSITION FROM Ready TO Busy
    := Do_;
END_TRANSITION
STEP Busy:
    Busy_active(N);  // step action
END_STEP
TRANSITION FROM Busy TO OpeningDoors2
    := DoWhat = 'CloseDoors' AND presence AND NOT Alt;
END_TRANSITION
STEP OpeningDoors2:
    Open_act(N);
END_STEP
TRANSITION FROM OpeningDoors2 TO Busy
    := Opened_sensor;
END_TRANSITION
TRANSITION FROM Busy TO ClosingDoors
    := DoWhat = 'CloseDoors' AND NOT Presence AND NOT Alt;
END_TRANSITION
STEP ClosingDoors:
    Close_act(N);
END_STEP
TRANSITION FROM ClosingDoors TO SetDone
    := NOT Presence AND Closed_sensor AND NOT Alt;
END_TRANSITION
TRANSITION FROM ClosingDoors TO OpeningDoors2
    := Presence AND NOT Alt;
END_TRANSITION
TRANSITION FROM ClosingDoors TO OpeningDoors
    := Alt;
END_TRANSITION
TRANSITION FROM Busy TO OpeningDoors
    := DoWhat = 'OpenDoors' OR Alt;
END_TRANSITION
STEP OpeningDoors:
    Open_act(N);
END_STEP
TRANSITION FROM OpeningDoors TO SetDone
    := Opened_sensor;
END_TRANSITION
STEP SetDone:
    Done(S);
END_STEP
TRANSITION FROM SetDone TO ResetDone
    := NOT Do_;
END_TRANSITION
STEP ResetDone:
    Done(R);
END_STEP
TRANSITION FROM ResetDone TO Ready
    := TRUE;
END_TRANSITION

ACTION Init_active:
State := 'Init';
END_ACTION

ACTION Ready_active:
State := 'Ready';
END_ACTION

ACTION Busy_active:
State := 'Busy';
END_ACTION

END_FUNCTION_BLOCK

// Device/Application/PLC_PRG
PROGRAM PLC_PRG
VAR
	Synchronization: BOOL;
	OperationOK: BOOL;
	
	UpExtCalls: ARRAY[0..6] OF BOOL;
	DownExtCalls: ARRAY[0..6] OF BOOL;
	IntCalls: ARRAY[0..7] OF BOOL;
	
	i: INT;
	B: INT;
	Up_dir: BOOL;
	Call: BOOL;
	NewDest: INT;
	DoubleChange: BOOL;
	CheckOpposite: BOOL;
	
	FaultSolved: BOOL;
	FaultD: BOOL;
	FaultR: BOOL;
	
	FaultLevelD: ARRAY[0..7] OF INT;
	FaultLevelR: ARRAY[0..7] OF INT;
END_VAR

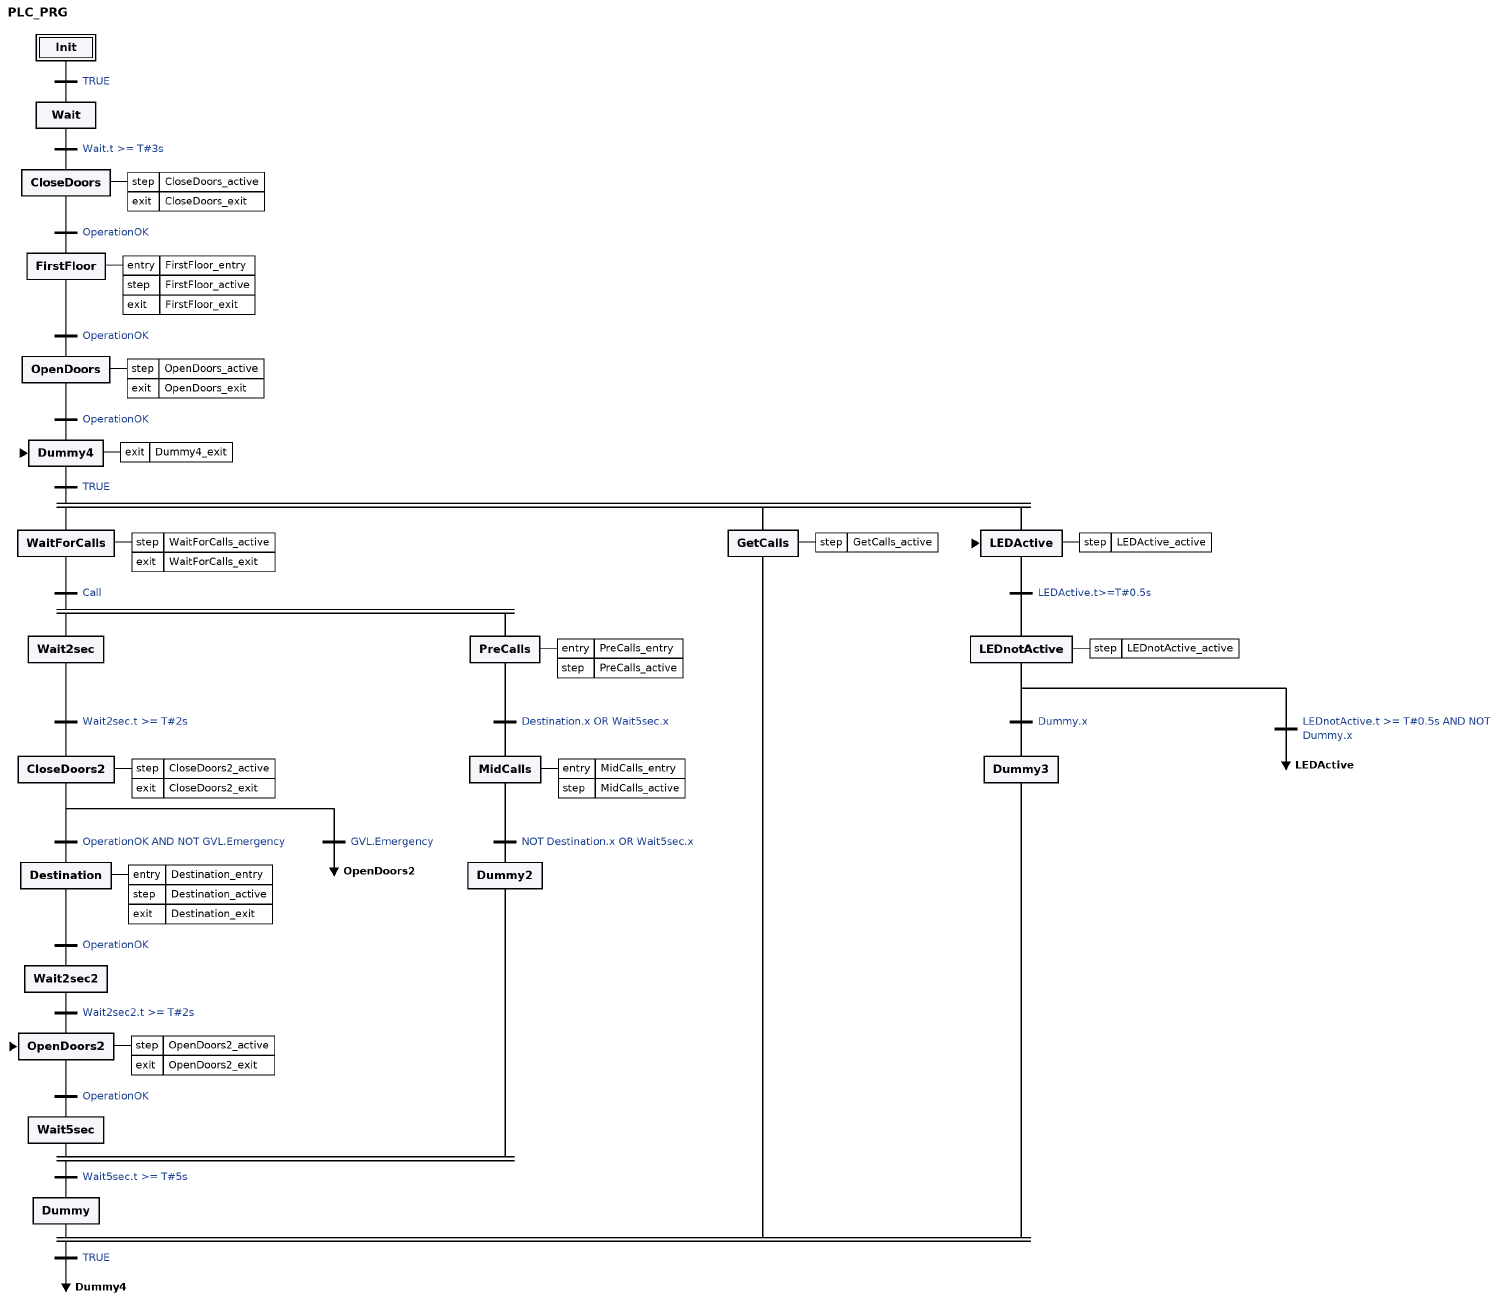
INITIAL_STEP Init:
END_STEP
TRANSITION FROM Init TO Wait
    := TRUE;
END_TRANSITION
STEP Wait:
END_STEP
TRANSITION FROM Wait TO CloseDoors
    := Wait.t >= T#3s;
END_TRANSITION
STEP CloseDoors:
    CloseDoors_active(N);  // step action
    CloseDoors_exit(P0);  // exit action
END_STEP
TRANSITION FROM CloseDoors TO FirstFloor
    := OperationOK;
END_TRANSITION
STEP FirstFloor:
    FirstFloor_entry(P1);  // entry action
    FirstFloor_active(N);  // step action
    FirstFloor_exit(P0);  // exit action
END_STEP
TRANSITION FROM FirstFloor TO OpenDoors
    := OperationOK;
END_TRANSITION
STEP OpenDoors:
    OpenDoors_active(N);  // step action
    OpenDoors_exit(P0);  // exit action
END_STEP
TRANSITION FROM OpenDoors TO Dummy4
    := OperationOK;
END_TRANSITION
STEP Dummy4:
    Dummy4_exit(P0);  // exit action
END_STEP
TRANSITION FROM Dummy4 TO (WaitForCalls, GetCalls, LEDActive)
    := TRUE;
END_TRANSITION
STEP WaitForCalls:
    WaitForCalls_active(N);  // step action
    WaitForCalls_exit(P0);  // exit action
END_STEP
TRANSITION FROM WaitForCalls TO (Wait2sec, PreCalls)
    := Call;
END_TRANSITION
STEP Wait2sec:
END_STEP
TRANSITION FROM Wait2sec TO CloseDoors2
    := Wait2sec.t >= T#2s;
END_TRANSITION
STEP CloseDoors2:
    CloseDoors2_active(N);  // step action
    CloseDoors2_exit(P0);  // exit action
END_STEP
TRANSITION FROM CloseDoors2 TO Destination
    := OperationOK AND NOT GVL.Emergency;
END_TRANSITION
TRANSITION FROM CloseDoors2 TO OpenDoors2
    := GVL.Emergency;
END_TRANSITION
STEP Destination:
    Destination_entry(P1);  // entry action
    Destination_active(N);  // step action
    Destination_exit(P0);  // exit action
END_STEP
TRANSITION FROM Destination TO Wait2sec2
    := OperationOK;
END_TRANSITION
STEP Wait2sec2:
END_STEP
TRANSITION FROM Wait2sec2 TO OpenDoors2
    := Wait2sec2.t >= T#2s;
END_TRANSITION
STEP OpenDoors2:
    OpenDoors2_active(N);  // step action
    OpenDoors2_exit(P0);  // exit action
END_STEP
TRANSITION FROM OpenDoors2 TO Wait5sec
    := OperationOK;
END_TRANSITION
STEP Wait5sec:
END_STEP
STEP PreCalls:
    PreCalls_entry(P1);  // entry action
    PreCalls_active(N);  // step action
END_STEP
TRANSITION FROM PreCalls TO MidCalls
    := Destination.x OR Wait5sec.x;
END_TRANSITION
STEP MidCalls:
    MidCalls_entry(P1);  // entry action
    MidCalls_active(N);  // step action
END_STEP
TRANSITION FROM MidCalls TO Dummy2
    := NOT Destination.x OR Wait5sec.x;
END_TRANSITION
STEP Dummy2:
END_STEP
TRANSITION FROM (Wait5sec, Dummy2) TO Dummy
    := Wait5sec.t >= T#5s;
END_TRANSITION
STEP Dummy:
END_STEP
STEP GetCalls:
    GetCalls_active(N);  // step action
END_STEP
STEP LEDActive:
    LEDActive_active(N);  // step action
END_STEP
TRANSITION FROM LEDActive TO LEDnotActive
    := LEDActive.t>=T#0.5s;
END_TRANSITION
STEP LEDnotActive:
    LEDnotActive_active(N);  // step action
END_STEP
TRANSITION FROM LEDnotActive TO Dummy3
    := Dummy.x;
END_TRANSITION
TRANSITION FROM LEDnotActive TO LEDActive
    := LEDnotActive.t >= T#0.5s AND NOT Dummy.x;
END_TRANSITION
STEP Dummy3:
END_STEP
TRANSITION FROM (Dummy, GetCalls, Dummy3) TO Dummy4
    := TRUE;
END_TRANSITION

ACTION Closing_active:
IF GVL.ManageDoors.State='Ready' THEN
	GVL.ManageDoors.Do_:=TRUE;
	GVL.ManageDoors.DoWhat:='CloseDoors';
END_IF

IF GVL.ManageDoors.State='Busy' AND GVL.ManageDoors.Done=TRUE THEN
	GVL.ManageDoors.Do_:=FALSE;
	Synchronization:=TRUE;
END_IF

OperationOK:= Synchronization AND NOT GVL.ManageDoors.Done;
END_ACTION

ACTION Closing_exit:
OperationOK:=FALSE;
Synchronization:=FALSE;
END_ACTION

ACTION CloseDoors2_exit:
OperationOK:=FALSE;
Synchronization:=FALSE;
END_ACTION

ACTION CloseDoors_active:
//If Doors_GA is Ready, the Policy sends a closing request
IF GVL.ManageDoors.State='Ready' THEN
	GVL.ManageDoors.Do_:=TRUE;
	GVL.ManageDoors.DoWhat:='CloseDoors'; 
END_IF

//If the operation is completed, the Policy can proceed
IF GVL.ManageDoors.State='Busy' AND GVL.ManageDoors.Done=TRUE THEN
	GVL.ManageDoors.Do_:=FALSE;
	Synchronization:=TRUE;
END_IF

OperationOK:= Synchronization AND NOT GVL.ManageDoors.Done;
END_ACTION

ACTION CloseDoors_exit:
OperationOK:=FALSE;
Synchronization:=FALSE;
END_ACTION

ACTION FirstFloor_active:
//If Motoring_GA is Ready, the Policy sends a Initialization request
IF GVL.Motoring.State='Ready' THEN
	GVL.Motoring.Do_:=TRUE;
	GVL.Motoring.DoWhat:='Initial';
END_IF

//Setting destination to First Floor, once Ground is reached
GVL.Motoring.GoTo := 1;
GVL.Motoring.GoFrom := 0;

//If the operation is completed, the Policy can proceed
IF GVL.Motoring.State='Busy' AND GVL.Motoring.Done=TRUE THEN
	GVL.Motoring.Do_:=FALSE;
	Synchronization:=TRUE;
END_IF

OperationOK:= Synchronization AND NOT GVL.Motoring.Done;
END_ACTION

ACTION FirstFloor_exit:
OperationOK:=FALSE;
Synchronization:=FALSE;

//Initializing Variables
GVL.Destination := GVL.Current;
IF GVL.Motoring.GoTo > GVL.Motoring.GoFrom THEN
	Up_dir := TRUE;
ELSE
	Up_dir := FALSE;
END_IF
DoubleChange := FALSE;
FaultSolved := FALSE;
FaultD := FALSE;
FaultR := FALSE;
FOR i:=0 TO 7 BY 1 DO
	FaultLevelD[i] := -1;
	FaultLevelR[i] := -1;
END_FOR
END_ACTION

ACTION OpenDoors_active:
//If Doors_GA is Ready, the Policy sends an opening request
IF GVL.ManageDoors.State='Ready' THEN
	GVL.ManageDoors.Do_:=TRUE;
	GVL.ManageDoors.DoWhat:='OpenDoors'; 
END_IF

//If the operation is completed, the Policy can proceed
IF GVL.ManageDoors.State='Busy' AND GVL.ManageDoors.Done=TRUE THEN
	GVL.ManageDoors.Do_:=FALSE;
	Synchronization:=TRUE;
END_IF

OperationOK:= Synchronization AND NOT GVL.ManageDoors.Done;
END_ACTION

ACTION OpenDoors_exit:
OperationOK:=FALSE;
Synchronization:=FALSE;
END_ACTION

ACTION CloseDoors2_active:
//If Doors_GA is Ready and there is no Emergency, the Policy sends a closing request
IF GVL.ManageDoors.State='Ready' AND NOT GVL.Emergency THEN
	GVL.ManageDoors.Do_:=TRUE;
	GVL.ManageDoors.DoWhat:='CloseDoors'; 
END_IF

//If the operation is completed, the Policy can proceed
IF GVL.ManageDoors.State='Busy' AND GVL.ManageDoors.Done=TRUE THEN
	GVL.ManageDoors.Do_:=FALSE;
	Synchronization:=TRUE;
END_IF

OperationOK:= Synchronization AND NOT GVL.ManageDoors.Done;
END_ACTION

ACTION Destination_active:
//If Motoring_GA is Ready, the Policy sends the DO request
IF GVL.Motoring.State='Ready' THEN
	GVL.Motoring.Do_:=TRUE;
	GVL.Motoring.DoWhat := 'Nominal';
	GVL.Motoring.GoFrom := GVL.Current;
END_IF

//Destinations can be changed, even when State is 'Busy'
GVL.Motoring.GoTo := GVL.Destination;
GVL.Motoring.GoToWanted := NewDest;

//If the GA grants the feasibility of the new destination, it is updated
IF GVL.Motoring.ChangeDest_Ok THEN
	GVL.Destination := NewDest;	
	GVL.Motoring.GoTo := NewDest;
END_IF

//EMERGENCY HANDLING
//In case of Emergency, the destination is changed to the nearest possible Floor 
IF GVL.Motoring.CheckAlt AND GVL.Emergency THEN
	GVL.Destination := GVL.Motoring.AltFloorFix;
	GVL.Motoring.GoTo := GVL.Motoring.AltFloorFix;	
END_IF

//If the operation is completed, the Policy can proceed
IF GVL.Motoring.State='Busy' AND GVL.Motoring.Done=TRUE THEN
	GVL.Motoring.Do_:=FALSE;
	Synchronization:=TRUE;
END_IF

OperationOK:= Synchronization AND NOT GVL.Motoring.Done;
END_ACTION

ACTION Destination_exit:
OperationOK:=FALSE;
Synchronization:=FALSE;

NewDest := -1;

//Reset Calls and Direction change
IF GVL.Current <> 7 AND Up_dir THEN
	IF (UpExtCalls[GVL.Current] = FALSE AND IntCalls[GVL.Current] = FALSE) THEN
		DownExtCalls[GVL.Current-1] := FALSE;
		Up_dir := FALSE;
	ELSIF UpExtCalls[GVL.Current] = TRUE THEN
		UpExtCalls[GVL.Current] := FALSE; //Remember UpExtCalls[GVL.Current] does not exist at 7th FLOOR
	END_IF
ELSIF Up_dir AND GVL.Current = 7 THEN
	DownExtCalls[GVL.Current-1] := FALSE;
	Up_dir := FALSE;
ELSIF GVL.Current <> 0 AND NOT Up_dir THEN
	IF (DownExtCalls[GVL.Current-1] = FALSE AND IntCalls[GVL.Current] = FALSE) THEN
		UpExtCalls[GVL.Current] := FALSE;
		Up_dir := TRUE;
	ELSIF DownExtCalls[GVL.Current-1] = TRUE THEN
		DownExtCalls[GVL.Current-1] := FALSE;
	END_IF
ELSIF NOT Up_dir AND GVL.Current = 0 THEN //Remember DownExtCalls[GVL.Current-1] does not exist at GROUND FLOOR
		UpExtCalls[GVL.Current] := FALSE;
		Up_dir := TRUE;
END_IF
IntCalls[GVL.Current] := FALSE; //Always reset Internal Panel Call

//FAULT HANDLING
//Deck/Ramp Faults values are stored for later uses
IF GVL.Motoring.FaultDeck THEN
	FaultD := TRUE;
END_IF
IF GVL.Motoring.FaultRamp THEN
	FaultR := TRUE;
END_IF
IF FaultLevelD[0] = -1 THEN
	FaultLevelD[0] := GVL.Motoring.FaultFloorD[0]; //Deck Fault Floor
END_IF
IF FaultLevelR[0] = -1 THEN
	FaultLevelR[0] := GVL.Motoring.FaultFloorR[0]; //Ramp Fault Floor (Up)
END_IF
IF FaultLevelR[1] = -1 THEN
	FaultLevelR[1] := GVL.Motoring.FaultFloorR[1]; //Ramp Fault Floor (Down)
END_IF

//Destination corrections - Faults
IF FaultR AND (GVL.Motoring.GoTo = FaultLevelR[0] OR GVL.Motoring.GoTo = FaultLevelR[1]) THEN
	GVL.Destination := GVL.Current;
END_IF
IF FaultD AND (GVL.Motoring.GoTo = FaultLevelD[0]) THEN
	GVL.Destination := GVL.Current;
END_IF

//Ramp Fault array assignement
GVL.Motoring.PrecFaultFlR := FaultLevelR;
END_ACTION

ACTION OpenDoors2_active:
//If Doors_GA is Ready, the Policy sends an opening request
IF GVL.ManageDoors.State='Ready' THEN
	GVL.ManageDoors.Do_:=TRUE;
	GVL.ManageDoors.DoWhat:='OpenDoors'; 
END_IF

//If the operation is completed, the Policy can proceed
IF GVL.ManageDoors.State='Busy' AND GVL.ManageDoors.Done=TRUE THEN
	GVL.ManageDoors.Do_:=FALSE;
	Synchronization:=TRUE;
END_IF

OperationOK:= Synchronization AND NOT GVL.ManageDoors.Done;
END_ACTION

ACTION OpenDoors2_exit:
OperationOK:=FALSE;
Synchronization:=FALSE;
END_ACTION

ACTION WaitForCalls_active:
//Finds the 'best' destination among the ones stored

// Variables Initialization
Call := FALSE;
CheckOpposite := FALSE;
B := -1;

//Check if any call is present, different from the one with a Deck Fault
FOR i := 0 TO 7 BY 1 DO //Checking calls of the Internal panel
	IF IntCalls[i] AND i <> FaultLevelD[0] THEN
		CheckOpposite := TRUE;
	END_IF
END_FOR

FOR i := 0 TO 6 BY 1 DO //Checking calls of the External panel (Up arrow)
	IF UpExtCalls[i] AND i <> FaultLevelD[0] THEN
		CheckOpposite := TRUE;
	END_IF
END_FOR

FOR i := 0 TO 6 BY 1 DO //Checking calls of the External panel (Down arrow)
	IF DownExtCalls[i] AND i+1 <> FaultLevelD[0] THEN
		CheckOpposite := TRUE;
	END_IF
END_FOR

//Algorithm that finds the best called destination
IF Up_dir AND CheckOpposite THEN
		
	//IF Elevator is going UPWARDS
	// -BEST CASE 1
	FOR i := 0 TO 7 BY 1 DO
		IF IntCalls[7-i] THEN
				IF (7-i) > GVL.Current AND (7-i) <> FaultLevelD[0] THEN 
					B := (7-i);
				END_IF
		END_IF
	END_FOR
	
	// -BEST CASE 2
	FOR i := 0 TO 6 BY 1 DO
		IF UpExtCalls[6-i] THEN
				IF (6-i) > GVL.Current AND ((6-i) < B OR B = -1) AND (6-i) <> FaultLevelD[0] THEN 
					B := (6-i);
				END_IF
		END_IF
	END_FOR
	
	// -MEDIUM CASE
	IF B = -1 THEN
		FOR i := 0 TO 6 BY 1 DO
			IF DownExtCalls[i] AND i+1 > GVL.Current AND i+1 <> FaultLevelD[0] THEN
				B := i + 1;
			END_IF
		END_FOR
	END_IF
	
	// -WORST CASE
	IF B = -1 THEN
		Up_dir := FALSE;
		DoubleChange := TRUE;
	END_IF
	
ELSIF NOT Up_dir AND CheckOpposite THEN
	
	//IF Elevator is going DOWNWARDS
	// -BEST CASE 1
	FOR i := 0 TO 7 BY 1 DO
		IF IntCalls[i] THEN
				IF i < GVL.Current  AND i <> FaultLevelD[0] THEN 
					B := i;
				END_IF
		END_IF
	END_FOR
	
	// -BEST CASE 2
	FOR i := 0 TO 6 BY 1 DO
		IF DownExtCalls[i] THEN
				IF i+1 < GVL.Current AND (i+1 > B OR B = -1) AND i+1 <> FaultLevelD[0] THEN 
					B := i+1;
				END_IF
		END_IF
	END_FOR
	
	// -MEDIUM CASE
	IF B = -1 THEN
		FOR i := 0 TO 6 BY 1 DO
			IF UpExtCalls[6-i] AND 6-i < GVL.Current AND 6-i <> FaultLevelD[0] THEN
				B := 6 - i;
			END_IF
		END_FOR
	END_IF
	
	// -WORST CASE
	IF B = -1 THEN
		Up_dir := TRUE;
		DoubleChange := TRUE;
	END_IF	
	
END_IF

//The best destination is given to GVL.Destination variable
IF  B <> -1 AND B <> GVL.Current AND NOT GVL.Emergency THEN
	Call := TRUE;
	GVL.Destination := B;
END_IF
END_ACTION

ACTION PreCalls_active:
//Finds if a possible NEW 'best' destination is called
//before the starting of the motor (with no restrictions in direction)

// Variables Initialization
Call := FALSE;
B := -1;

//Check if any NEW call is present, different from the one already considered
//and, if present, different from the one with a Deck Fault
FOR i := 0 TO 7 BY 1 DO
	IF IntCalls[i] AND i <> GVL.Destination AND i <> FaultLevelD[0] THEN
		Call := TRUE;
	END_IF
END_FOR

FOR i := 0 TO 6 BY 1 DO
	IF UpExtCalls[i] AND i <> GVL.Destination AND i <> FaultLevelD[0] THEN
		Call := TRUE;
	END_IF
END_FOR

FOR i := 0 TO 6 BY 1 DO
	IF DownExtCalls[i] AND i+1 <> GVL.Destination AND i+1 <> FaultLevelD[0] THEN
		Call := TRUE;
	END_IF
END_FOR

//Algorithm that finds the best called destination
IF Up_dir AND Call THEN
		
	//IF Elevator is going UPWARDS
	// -BEST CASE 1
	FOR i := 0 TO 7 BY 1 DO
		IF IntCalls[7-i] THEN
				IF (7-i) > GVL.Current AND (7-i) <> FaultLevelD[0] THEN 
					B := (7-i);
				END_IF
		END_IF
	END_FOR
	
	// -BEST CASE 2
	FOR i := 0 TO 6 BY 1 DO
		IF UpExtCalls[6-i] THEN
				IF (6-i) > GVL.Current AND ((6-i) < B OR B = -1) AND (6-i) <> FaultLevelD[0] THEN 
					B := (6-i);
				END_IF
		END_IF
	END_FOR
	
	// -MEDIUM CASE
	IF B = -1 THEN
		FOR i := 0 TO 6 BY 1 DO
			IF DownExtCalls[i] AND i+1 > GVL.Current AND i+1 <> FaultLevelD[0] THEN
				B := i + 1;
			END_IF
		END_FOR
	END_IF
	
	// -WORST CASE
	IF B = -1 AND CheckOpposite THEN
		Up_dir := FALSE;
	END_IF	
	
ELSE
	//IF Elevator is going DOWNWARDS
	// -BEST CASE 1
	FOR i := 0 TO 7 BY 1 DO
		IF IntCalls[i] THEN
				IF i < GVL.Current AND i <> FaultLevelD[0] THEN 
					B := i;
				END_IF
		END_IF
	END_FOR
	
	// -BEST CASE 2
	FOR i := 0 TO 6 BY 1 DO
		IF DownExtCalls[i] THEN
				IF i+1 < GVL.Current AND (i+1 > B OR B = -1) AND i+1 <> FaultLevelD[0] THEN 
					B := i+1;
				END_IF
		END_IF
	END_FOR
	
	// -MEDIUM CASE
	IF B = -1 THEN
		FOR i := 0 TO 6 BY 1 DO
			IF UpExtCalls[6-i] AND 6-i < GVL.Current AND 6-i <> FaultLevelD[0] THEN
				B := 6 - i;
			END_IF
		END_FOR
	END_IF
	
	// -WORST CASE
	IF B = -1 AND CheckOpposite THEN
		Up_dir := TRUE;
	END_IF	
	
END_IF

//If a NEW destination, better from the already considered one, is found
//it is assigned to GVL.Destination variable
IF  B <> -1 AND B <> GVL.Destination AND B <> GVL.Current AND NOT GVL.Emergency THEN
	GVL.Destination := B;
END_IF
END_ACTION

ACTION MidCalls_active:
//Finds if a possible NEW 'best' destination is called
//after the starting of the motor (with obvious restrictions in direction)

// Variables Initialization
Call := FALSE;
B := -1;

//Check if any NEW call is present, different from the one already considered
//and, if present, different from the one with a Deck Fault
FOR i := 0 TO 7 BY 1 DO
	IF IntCalls[i] AND i <> GVL.Destination AND i <> FaultLevelD[0]THEN
		Call := TRUE;
	END_IF
END_FOR

FOR i := 0 TO 6 BY 1 DO
	IF UpExtCalls[i] AND i <> GVL.Destination AND i <> FaultLevelD[0] THEN
		Call := TRUE;
	END_IF
END_FOR

FOR i := 0 TO 6 BY 1 DO
	IF DownExtCalls[i] AND i+1 <> GVL.Destination AND i+1 <> FaultLevelD[0] THEN
		Call := TRUE;
	END_IF
END_FOR

//The direction cannot be changed anymore (since the motor is already ON) 
IF GVL.Destination > GVL.Current THEN
	Up_dir := TRUE;
ELSIF GVL.Destination < GVL.Current THEN
	Up_dir := FALSE; 
END_IF

//Algorithm that finds the best called destination
//WORST CASEs are no longered taken into account 
IF Up_dir AND Call THEN
	
	//IF Elevator is going UPWARDS
	// -BEST CASE 1
	FOR i := 0 TO 7 BY 1 DO
		IF IntCalls[7-i] THEN
				IF (7-i) > GVL.Current AND (7-i) <> FaultLevelD[0] THEN 
					B := (7-i);
				END_IF
		END_IF
	END_FOR
	
	// -BEST CASE 2
	FOR i := 0 TO 6 BY 1 DO
		IF UpExtCalls[6-i] THEN
				IF (6-i) > GVL.Current AND ((6-i) < B OR B = -1) AND (6-i) <> FaultLevelD[0] THEN 
					B := (6-i);
				END_IF
		END_IF
	END_FOR
	
	// -MEDIUM CASE
	IF B = -1 THEN
		FOR i := 0 TO 6 BY 1 DO
			IF DownExtCalls[i] AND i+1 > GVL.Current AND i+1 <> FaultLevelD[0] THEN
				B := i + 1;
			END_IF
		END_FOR
	END_IF	
	
ELSE
	//IF Elevator is going DOWNWARDS
	// -BEST CASE 1
	FOR i := 0 TO 7 BY 1 DO
		IF IntCalls[i] THEN
				IF i < GVL.Current AND i <> FaultLevelD[0] THEN 
					B := i;
				END_IF
		END_IF
	END_FOR
	
	// -BEST CASE 2
	FOR i := 0 TO 6 BY 1 DO
		IF DownExtCalls[i] THEN
				IF i+1 < GVL.Current AND (i+1 > B OR B = -1) AND i+1 <> FaultLevelD[0] THEN 
					B := i+1;
				END_IF
		END_IF
	END_FOR
	
	// -MEDIUM CASE
	IF B = -1 THEN
		FOR i := 0 TO 6 BY 1 DO
			IF UpExtCalls[6-i] AND 6-i < GVL.Current AND 6-i <> FaultLevelD[0] THEN
				B := 6 - i;
			END_IF
		END_FOR
	END_IF
	
END_IF

//If a NEW destination, better from the already considered one, is found
//it is assigned to NewDest variable
//NewDest is then sent to the Motoring_GA, which checks its feasibility
IF  B <> -1 AND B <> GVL.Destination AND B <> GVL.Current AND NOT GVL.Emergency THEN
	NewDest := B;
END_IF
END_ACTION

ACTION MidCalls_entry:
//Initialization of NewDest
NewDest := -1;
END_ACTION

ACTION WaitForCalls_exit:
NewDest := -1;
END_ACTION

ACTION PreCalls_entry:
//If DoubleChange is TRUE, direction was changed in the WaitForCalls block
//If new calls in the original direction are made, they will be preferred
//Here the direction is reversed so that such calls are given priority
IF DoubleChange THEN
	IF Up_dir THEN
		Up_dir := FALSE;
	ELSE 
		Up_dir := TRUE;
	END_IF
END_IF
END_ACTION

ACTION Dummy4_exit:
DoubleChange := FALSE;
END_ACTION

ACTION LEDActive_active:
//If there is a Deck Fault, the corresponding Floor Arrows flash alternatively
IF FaultLevelD[0] <> -1 AND FaultD THEN
	CASE FaultLevelD[0] OF
		0: GVL.UpDeckGVis := TRUE;
		   GVL.PGVis := TRUE;
		1: GVL.UpDeck1Vis := TRUE;
		   GVL.DownDeck1Vis := FALSE;
		   GVL.P1Vis := TRUE;
		2: GVL.UpDeck2Vis := TRUE;
		   GVL.DownDeck2Vis := FALSE;
		   GVL.P2Vis := TRUE;
		3: GVL.UpDeck3Vis := TRUE;
		   GVL.DownDeck3Vis := FALSE;
		   GVL.P3Vis := TRUE;
		4: GVL.UpDeck4Vis := TRUE;
		   GVL.DownDeck4Vis := FALSE;
		   GVL.P4Vis := TRUE;
		5: GVL.UpDeck5Vis := TRUE;
		   GVL.DownDeck5Vis := FALSE;
		   GVL.P5Vis := TRUE;
		6: GVL.UpDeck6Vis := TRUE;
		   GVL.DownDeck6Vis := FALSE;
		   GVL.P6Vis := TRUE;
		7: GVL.DownDeck7Vis := FALSE;
		   GVL.P7Vis := TRUE;
	END_CASE
END_IF
END_ACTION

ACTION LEDnotActive_active:
//If there is a Deck Fault, the corresponding Floor Arrows flash alternatively
IF FaultLevelD[0] <> -1 AND FaultD THEN
	CASE FaultLevelD[0] OF
		0: GVL.UpDeckGVis := FALSE;
		   GVL.PGVis := FALSE;
		1: GVL.UpDeck1Vis := FALSE;
		   GVL.DownDeck1Vis := TRUE;
		   GVL.P1Vis := FALSE;
		2: GVL.UpDeck2Vis := FALSE;
		   GVL.DownDeck2Vis := TRUE;
		   GVL.P2Vis := FALSE;
		3: GVL.UpDeck3Vis := FALSE;
		   GVL.DownDeck3Vis := TRUE;
		   GVL.P3Vis := FALSE;
		4: GVL.UpDeck4Vis := FALSE;
		   GVL.DownDeck4Vis := TRUE;
		   GVL.P4Vis := FALSE;
		5: GVL.UpDeck5Vis := FALSE;
		   GVL.DownDeck5Vis := TRUE;
		   GVL.P5Vis := FALSE;
		6: GVL.UpDeck6Vis := FALSE;
		   GVL.DownDeck6Vis := TRUE;
		   GVL.P6Vis := FALSE;
		7: GVL.DownDeck7Vis := TRUE;
		   GVL.P7Vis := FALSE;
	END_CASE
END_IF
END_ACTION

ACTION GetCalls_active:
//Looking and storing Calls

//Calls from External Panel (Up arrow)
IF NOT UpExtCalls[0] THEN
	UpExtCalls[0] := GVL.UpDeckG;
END_IF
IF NOT UpExtCalls[1] THEN
	UpExtCalls[1] := GVL.UpDeck1;
END_IF
IF NOT UpExtCalls[2] THEN
	UpExtCalls[2] := GVL.UpDeck2;
END_IF
IF NOT UpExtCalls[3] THEN
	UpExtCalls[3] := GVL.UpDeck3;
END_IF
IF NOT UpExtCalls[4] THEN
	UpExtCalls[4] := GVL.UpDeck4;
END_IF
IF NOT UpExtCalls[5] THEN
	UpExtCalls[5] := GVL.UpDeck5;
END_IF
IF NOT UpExtCalls[6] THEN
	UpExtCalls[6] := GVL.UpDeck6;
END_IF

//Calls from External Panel (Down arrow)
IF NOT DownExtCalls[0] THEN
	DownExtCalls[0] := GVL.DownDeck1;
END_IF
IF NOT DownExtCalls[1] THEN
	DownExtCalls[1] := GVL.DownDeck2;
END_IF
IF NOT DownExtCalls[2] THEN
	DownExtCalls[2] := GVL.DownDeck3;
END_IF
IF NOT DownExtCalls[3] THEN
	DownExtCalls[3] := GVL.DownDeck4;
END_IF
IF NOT DownExtCalls[4] THEN
	DownExtCalls[4] := GVL.DownDeck5;
END_IF
IF NOT DownExtCalls[5] THEN
	DownExtCalls[5] := GVL.DownDeck6;
END_IF
IF NOT DownExtCalls[6] THEN
	DownExtCalls[6] := GVL.DownDeck7;
END_IF

//Calls from Internal Panel (different from Current Floor)
IF NOT IntCalls[0] AND GVL.Current <> 0 THEN
	IntCalls[0] := GVL.PG;
END_IF
IF NOT IntCalls[1] AND GVL.Current <> 1 THEN
	IntCalls[1] := GVL.P1;
END_IF
IF NOT IntCalls[2] AND GVL.Current <> 2 THEN
	IntCalls[2] := GVL.P2;
END_IF
IF NOT IntCalls[3] AND GVL.Current <> 3 THEN
	IntCalls[3] := GVL.P3;
END_IF
IF NOT IntCalls[4] AND GVL.Current <> 4 THEN
	IntCalls[4] := GVL.P4;
END_IF
IF NOT IntCalls[5] AND GVL.Current <> 5 THEN
	IntCalls[5] := GVL.P5;
END_IF
IF NOT IntCalls[6] AND GVL.Current <> 6 THEN
	IntCalls[6] := GVL.P6;
END_IF
IF NOT IntCalls[7] AND GVL.Current <> 7 THEN
	IntCalls[7] := GVL.P7;
END_IF

//LEDs Handling
GVL.UpDeckGVis := UpExtCalls[0];
GVL.UpDeck1Vis := UpExtCalls[1];
GVL.UpDeck2Vis := UpExtCalls[2];
GVL.UpDeck3Vis := UpExtCalls[3];
GVL.UpDeck4Vis := UpExtCalls[4];
GVL.UpDeck5Vis := UpExtCalls[5];
GVL.UpDeck6Vis := UpExtCalls[6];

GVL.DownDeck1Vis := DownExtCalls[0];
GVL.DownDeck2Vis := DownExtCalls[1];
GVL.DownDeck3Vis := DownExtCalls[2];
GVL.DownDeck4Vis := DownExtCalls[3];
GVL.DownDeck5Vis := DownExtCalls[4];
GVL.DownDeck6Vis := DownExtCalls[5];
GVL.DownDeck7Vis := DownExtCalls[6];

GVL.PGVis := IntCalls[0];
GVL.P1Vis := IntCalls[1];
GVL.P2Vis := IntCalls[2];
GVL.P3Vis := IntCalls[3];
GVL.P4Vis := IntCalls[4];
GVL.P5Vis := IntCalls[5];
GVL.P6Vis := IntCalls[6];
GVL.P7Vis := IntCalls[7];

//System Communications Panel Handling
GVL.EmergencyVis:= GVL.Emergency OR FaultD OR FaultR;
GVL.FaultSensorAlarm := FaultD;
GVL.FaultRampAlarm := FaultR;

//'Virtually' Solving Faults by pressing two times the Emergency Button
IF GVL.Emergency AND (FaultD OR FaultR) THEN
	FaultSolved := TRUE;
END_IF

IF FaultSolved AND NOT GVL.Emergency THEN
	FaultSolved := FALSE;
	FaultD := FALSE;
	FaultR := FALSE;
	FaultLevelD[0] := -1;
	FaultLevelR[0] := -1;
	FaultLevelR[1] := -1;
	GVL.Motoring.PrecFaultFlR := FaultLevelR;
END_IF
END_ACTION

ACTION FirstFloor_entry:
//Needed initialization variable
GVL.Motoring.GoToWanted := -1;
//Needed initialization array
FOR i:=0 TO 7 BY 1 DO
	FaultLevelR[i] := -1;
END_FOR
//Ramp Fault array assignement
GVL.Motoring.PrecFaultFlR := FaultLevelR;
END_ACTION

ACTION Destination_entry:
//Reset CALLS that changed the direction unexpectedly
IF Up_dir AND GVL.Current <> 7 THEN
	IF UpExtCalls[GVL.Current] THEN
		UpExtCalls[GVL.Current] := FALSE;
	END_IF
ELSIF NOT Up_dir AND GVL.Current <> 0 THEN
	IF DownExtCalls[GVL.Current-1] THEN
		DownExtCalls[GVL.Current-1] := FALSE;
	END_IF
END_IF
END_ACTION

END_PROGRAM

// Device/Application/Visualization
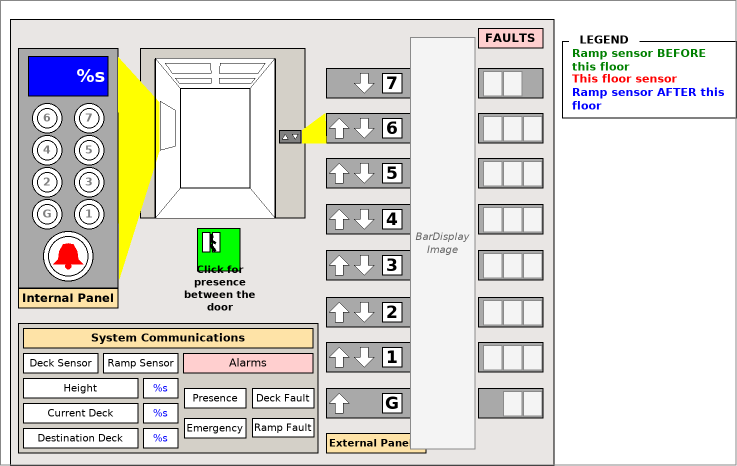
VISUALIZATION Visualization  // 737x466
    Rectangle (10,19 544x447)
    Rectangle (197,228 43x43), colour toggle: GVL.Presence
    Rectangle (18,323 300x130)
    Rectangle (326,433 100x20), "External Panels"
    Rectangle (326,342 100x30)
    Rectangle (382,347 20x20), "1"
    Polygon (354,357) (360,357) (360,347) (368,347) (368,357) (374,357) (364,367), colour toggle: GVL.DownDeck1Vis
        tap GVL.DownDeck1
    Polygon (329,357) (335,357) (335,367) (343,367) (343,357) (349,357) (339,347), colour toggle: GVL.UpDeck1Vis
        tap GVL.UpDeck1
    Rectangle (326,297 100x30)
    Rectangle (382,302 20x20), "2"
    Polygon (354,312) (360,312) (360,302) (368,302) (368,312) (374,312) (364,322), colour toggle: GVL.DownDeck2Vis
        tap GVL.DownDeck2
    Polygon (329,312) (335,312) (335,322) (343,322) (343,312) (349,312) (339,302), colour toggle: GVL.UpDeck2Vis
        tap GVL.UpDeck2
    Rectangle (326,250 100x30)
    Rectangle (382,255 20x20), "3"
    Polygon (354,265) (360,265) (360,255) (368,255) (368,265) (374,265) (364,275), colour toggle: GVL.DownDeck3Vis
        tap GVL.DownDeck3
    Polygon (329,265) (335,265) (335,275) (343,275) (343,265) (349,265) (339,255), colour toggle: GVL.UpDeck3Vis
        tap GVL.UpDeck3
    Rectangle (326,204 100x30)
    Rectangle (382,209 20x20), "4"
    Polygon (354,219) (360,219) (360,209) (368,209) (368,219) (374,219) (364,229), colour toggle: GVL.DownDeck4Vis
        tap GVL.DownDeck4
    Polygon (329,219) (335,219) (335,229) (343,229) (343,219) (349,219) (339,209), colour toggle: GVL.UpDeck4Vis
        tap GVL.UpDeck4
    Rectangle (326,158 100x30)
    Rectangle (382,163 20x20), "5"
    Polygon (354,173) (360,173) (360,163) (368,163) (368,173) (374,173) (364,183), colour toggle: GVL.DownDeck5Vis
        tap GVL.DownDeck5
    Polygon (329,173) (335,173) (335,183) (343,183) (343,173) (349,173) (339,163), colour toggle: GVL.UpDeck5Vis
        tap GVL.UpDeck5
    Rectangle (326,113 100x30)
    Rectangle (382,118 20x20), "6"
    Polygon (354,128) (360,128) (360,118) (368,118) (368,128) (374,128) (364,138), colour toggle: GVL.DownDeck6Vis
        tap GVL.DownDeck6
    Polygon (329,128) (335,128) (335,138) (343,138) (343,128) (349,128) (339,118), colour toggle: GVL.UpDeck6Vis
        tap GVL.UpDeck6
    Rectangle (326,68 100x30)
    Rectangle (382,73 20x20), "7"
    Polygon (354,83) (360,83) (360,73) (368,73) (368,83) (374,83) (364,93), colour toggle: GVL.DownDeck7Vis
        tap GVL.DownDeck7
    Rectangle (326,388 100x30)
    Rectangle (382,393 20x20), "G"
    Polygon (329,403) (335,403) (335,413) (343,413) (343,403) (349,403) (339,393), colour toggle: GVL.UpDeckGVis
        tap GVL.UpDeckG
    RoundedRectangle (18,48 100x240)
    Rectangle (18,288 100x20), "Internal Panel"
    Ellipse (74,199 30x30), colour toggle: GVL.P1Vis
    Ellipse (79,204 20x20), "1"
        tap GVL.P1
    Ellipse (32,199 30x30), colour toggle: GVL.PGVis
    Ellipse (37,204 20x20), "G"
        tap GVL.PG
    Ellipse (74,167 30x30), colour toggle: GVL.P3Vis
    Ellipse (79,172 20x20), "3"
        tap GVL.P3
    Ellipse (32,167 30x30), colour toggle: GVL.P2Vis
    Ellipse (37,172 20x20), "2"
        tap GVL.P2
    Ellipse (74,135 30x30), colour toggle: GVL.P5Vis
    Ellipse (79,140 20x20), "5"
        tap GVL.P5
    Ellipse (32,135 30x30), colour toggle: GVL.P4Vis
    Ellipse (37,140 20x20), "4"
        tap GVL.P4
    Ellipse (74,103 30x30), colour toggle: GVL.P7Vis
    Ellipse (79,108 20x20), "7"
        tap GVL.P7
    Ellipse (32,103 30x30), colour toggle: GVL.P6Vis
    Ellipse (37,108 20x20), "6"
        tap GVL.P6
    Rectangle (28,56 80x40), "%s", text variable: GVL.Destination
    Ellipse (43,231 50x50), tooltip "EMERGENCY", colour toggle: GVL.Emergency
    Group (48,236 40x40)
        toggle GVL.Emergency
        Ellipse (0,0 40x40), tooltip "EMERGENCY"
        Polygon (5,28) (10,23) (11,15) (15,8) (20,7) (25,8) (29,15) (30,23) (35,28)
        Ellipse (17,27 6x6)
    Polygon (35,72) (45,62) (55,72), colour toggle: GVL.Motor_on AND GVL.Up
    Polygon (35,80) (45,90) (55,80), colour toggle: GVL.Motor_on AND NOT GVL.Up
    Group (140,48 165x170)
        Rectangle (0,0 165x170)
        Rectangle (15,10 120x160)
        Polygon (40,40) (15,10) (135,10) (110,40)
        Rectangle (40,40 70x100)
        Polygon (15,170) (40,140) (110,140) (135,170)
        Polygon (20,102) (20,53) (35,62) (35,98)
        Polygon (79,35) (79,30) (115,30) (111,35)
        Polygon (39,35) (35,30) (71,30) (71,35)
        Polygon (32,25) (25,15) (70,15) (71,25)
        Polygon (79,25) (80,15) (125,15) (118,25)
        Group (139,82 22x13)
            Rectangle (0,0 22x13)
            Polygon (3,9) (6,4) (9,9)
            Polygon (13,4) (16,9) (19,4)
    BarDisplayImage (410,37 65x412), value: GVL.Height, style: BarDisplayImage-Gray, scale format: %.0f, scale -20..160
        p3451962224: VisuNativeControl.IP_Offline.Browser
    Rectangle (478,68 65x30)
    Rectangle (478,342 65x30)
    Rectangle (478,297 65x30)
    Rectangle (478,250 65x30)
    Rectangle (478,204 65x30)
    Rectangle (478,158 65x30)
    Rectangle (478,113 65x30)
    Rectangle (478,388 65x30)
    RockerSwitch (483,345 19x25), variable: GVL.Ramp1Down, behaviour: TOGGLE, style: Switch-RockerSwitch-Green
    RockerSwitch (503,345 19x25), variable: GVL.Sensor1, behaviour: TOGGLE, style: Switch-RockerSwitch-Red
    RockerSwitch (523,345 19x25), variable: GVL.Ramp1Up, behaviour: TOGGLE, style: Switch-RockerSwitch-Blue
    RockerSwitch (483,300 19x25), variable: GVL.Ramp2Down, behaviour: TOGGLE, style: Switch-RockerSwitch-Green
    RockerSwitch (503,300 19x25), variable: GVL.Sensor2, behaviour: TOGGLE, style: Switch-RockerSwitch-Red
    RockerSwitch (523,300 19x25), variable: GVL.Ramp2Up, behaviour: TOGGLE, style: Switch-RockerSwitch-Blue
    RockerSwitch (483,253 19x25), variable: GVL.Ramp3Down, behaviour: TOGGLE, style: Switch-RockerSwitch-Green
    RockerSwitch (503,253 19x25), variable: GVL.Sensor3, behaviour: TOGGLE, style: Switch-RockerSwitch-Red
    RockerSwitch (523,253 19x25), variable: GVL.Ramp3Up, behaviour: TOGGLE, style: Switch-RockerSwitch-Blue
    RockerSwitch (483,207 19x25), variable: GVL.Ramp4Down, behaviour: TOGGLE, style: Switch-RockerSwitch-Green
    RockerSwitch (503,207 19x25), variable: GVL.Sensor4, behaviour: TOGGLE, style: Switch-RockerSwitch-Red
    RockerSwitch (523,207 19x25), variable: GVL.Ramp4Up, behaviour: TOGGLE, style: Switch-RockerSwitch-Blue
    RockerSwitch (483,161 19x25), variable: GVL.Ramp5Down, behaviour: TOGGLE, style: Switch-RockerSwitch-Green
    RockerSwitch (503,161 19x25), variable: GVL.Sensor5, behaviour: TOGGLE, style: Switch-RockerSwitch-Red
    RockerSwitch (523,161 19x25), variable: GVL.Ramp5Up, behaviour: TOGGLE, style: Switch-RockerSwitch-Blue
    RockerSwitch (483,116 19x25), variable: GVL.Ramp6Down, behaviour: TOGGLE, style: Switch-RockerSwitch-Green
    RockerSwitch (503,116 19x25), variable: GVL.Sensor6, behaviour: TOGGLE, style: Switch-RockerSwitch-Red
    RockerSwitch (523,116 19x25), variable: GVL.Ramp6Up, behaviour: TOGGLE, style: Switch-RockerSwitch-Blue
    RockerSwitch (483,71 19x25), variable: GVL.Ramp7Down, behaviour: TOGGLE, style: Switch-RockerSwitch-Green
    RockerSwitch (503,71 19x25), variable: GVL.Sensor7, behaviour: TOGGLE, style: Switch-RockerSwitch-Red
    RockerSwitch (503,391 19x25), variable: GVL.SensorG, behaviour: TOGGLE, style: Switch-RockerSwitch-Red
    RockerSwitch (523,391 19x25), variable: GVL.RampGUp, behaviour: TOGGLE, style: Switch-RockerSwitch-Blue
    Rectangle (478,28 65x20), "FAULTS"
    Polygon (302,130) (325,113) (326,143) (302,143), invisible if: (GVL.Closing OR GVL.Opening) OR GVL.Closed
    Polygon (118,57) (159,102) (159,151) (119,279), invisible if: (GVL.Closing OR GVL.Opening) OR GVL.Closed
    Rectangle (155,58 0x160)
        p3528305787: GVL.Door
    Rectangle (275,58 0x160)
        p3528305787: -GVL.Door
    Rectangle (23,328 290x20), "System Communications"
    Rectangle (183,353 130x20), "Alarms"
    Rectangle (23,353 75x20), "Deck Sensor", colour toggle: GVL.DeckSensor
    Rectangle (143,378 35x20), "%s", text variable: GVL.Height
    Rectangle (184,388 62x20), "Presence", colour toggle: GVL.Presence
    Rectangle (103,353 75x20), "Ramp Sensor", colour toggle: GVL.RampSensor
    Rectangle (143,403 35x20), "%s", text variable: GVL.Current
    Rectangle (143,428 35x20), "%s", text variable: GVL.Destination
    Rectangle (252,388 62x20), "Deck Fault", colour toggle: GVL.FaultSensorAlarm
    Rectangle (184,418 62x20), "Emergency", colour toggle: GVL.EmergencyVis
    Rectangle (252,418 62x19), "Ramp Fault", colour toggle: GVL.FaultRampAlarm
    Rectangle (23,378 115x20), "Height"
    Rectangle (23,403 115x20), "Current Deck"
    Rectangle (23,428 115x20), "Destination Deck"
    Group (562,25 175x93)
        Rectangle (0,16 175x77)
        Rectangle (7,39 160x30), "This floor sensor"
        Rectangle (7,59 160x30), "Ramp sensor AFTER this floor"
        Rectangle (7,0 70x30), "LEGEND"
        Rectangle (7,20 160x30), "Ramp sensor BEFORE this floor"
    Group (202,232 33x34)
        toggle GVL.Presence
        Rectangle (10,0 8x20)
        Polygon (5,10) (12,20) (14,18) (5,6)
        Ellipse (6,2 5x5)
        Polygon (4,8) (13,12) (14,10) (4,4)
        Rectangle (0,0 8x20)
    Rectangle (169,273 102x31), "Click for presence between the door"
END_VISUALIZATION
